DATA_BLOCK "BRITADORES_DB"
{ S7_Optimized_Access := 'TRUE' }
VERSION : 0.1
NON_RETAIN
"BRITADORES"

BEGIN

END_DATA_BLOCK